TYPE Joint :
STRUCT
	position : INT;
END_STRUCT
END_TYPE

(* stored: Version 1.1.0.1, ProductVersion 3.1.4024.12
   DUT Joint: Id {ba4bf0d8-7ccb-42b6-ac15-60a638e315a7} *)
